TYPE ST_TsConnectionInfo1Byte :
(*******************************************************************************************************
Description			:	Connection information data of EtherCAT Slaves with 1 byte safe data 
Supported terminals : 	EL1904, EL2904...
Date 				:	04.04.2016
********************************************************************************************************)
STRUCT

	nState 	 								:USINT;
	nDiag 		 							:USINT;
	nInOutSafeDataByte1						:BYTE;
	
END_STRUCT
END_TYPE
(* End *)

(* stored: Version 1.1.0.1, ProductVersion 3.1.4022.16
   DUT ST_TsConnectionInfo1Byte: Id {f792b008-d0b3-4b22-8812-3b6a691e3a12} *)
